// TIA Portal V16 export
// export: Created 2021-07-12T14:47:15.2161229Z, ExportSetting WithDefaults, DisplayName Totally Integrated Automation Portal, DisplayVersion V16, DisplayName TIA Portal Version Control Interface, DisplayVersion V16, DisplayName TIA Portal Openness, DisplayVersion V16, DisplayName STEP 7 Professional, DisplayVersion V16, DisplayName STEP 7 Safety, DisplayVersion V16, DisplayName WinCC Professional, DisplayVersion V16
DATA_BLOCK "SimaHydTO_VCharArray"   // DB33102
TITLE = SimaHydTO_VCharArray
{ S7_Optimized_Access := 'TRUE'; DB_Accessible_From_OPC_UA := 'FALSE' }
FAMILY : SimaHydTO
VERSION : 1.0
// Array of valve chracteristics usabel in HMI
// stored: AutoNumber true, DBAccessibleFromOPCUA false, IsOnlyStoredInLoadMemory false, IsRetainMemResEnabled false, IsWriteProtectedInAS false, MemoryReserve 100
   VAR
      VChar { S7_SetPoint := 'True'} : Array[0..12] of "SimaHydTO_typeVCharArray";   // Valve charactersitics of the project to be controlled via HMI
   END_VAR
BEGIN
   VChar[0].VChar_DB := 5001;
END_DATA_BLOCK
